FUNCTION_BLOCK PedLightCtl (* Function block for controling the operation of a pedestrian trafic light with one red and one green light *)
  (* Standard: 61499-2 *)
  (* Version 0.0, 2014-07-11, 4DIAC-IDE, 4DIAC-Consortium *)
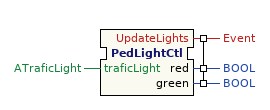
  EVENT_OUTPUT
    UpdateLights WITH green, red;
  END_EVENT
  VAR_OUTPUT
    red : BOOL;
    green : BOOL;
  END_VAR
  SOCKETS
    traficLight : ATraficLight;
  END_SOCKETS
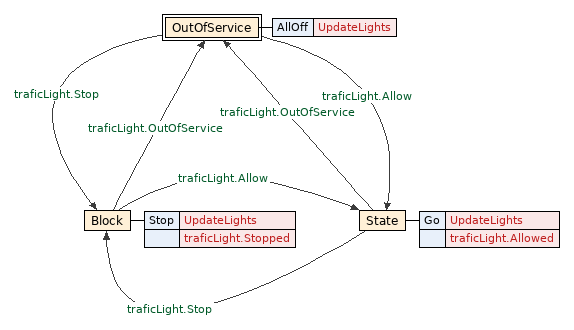
  EC_STATES
    OutOfService : AllOff -> UpdateLights;
    Block : Stop -> UpdateLights, -> traficLight.Stopped;
    State : Go -> UpdateLights, -> traficLight.Allowed;
  END_STATES
  EC_TRANSITIONS
    OutOfService TO Block := traficLight.Stop;
    Block TO OutOfService := traficLight.OutOfService;
    Block TO State := traficLight.Allow;
    State TO Block := traficLight.Stop;
    State TO OutOfService := traficLight.OutOfService;
    OutOfService TO State := traficLight.Allow;
  END_TRANSITIONS
  ALGORITHM AllOff IN ST:
red := FALSE;
green := FALSE;
  END_ALGORITHM
  ALGORITHM Stop IN ST: (* Put lights in stop mode (i.e., red := true, green := false) *)
red := TRUE;
green := FALSE;
  END_ALGORITHM
  ALGORITHM Go IN ST: (* Put lights in Walk mode (i.e., red := false, green := true) *)
red := FALSE;
green := TRUE;
  END_ALGORITHM
END_FUNCTION_BLOCK
